INTERFACE I_Singleton

METHOD Message : String
VAR_INPUT
END_VAR
END_METHOD

END_INTERFACE

(* stored: Version 1.1.0.1, ProductVersion 3.1.4024.12
   Itf I_Singleton: Id {a5eba910-5db8-4f2d-a1d3-8e1dad0343dd}
   Method Message: Id {d8f90746-29e8-4fd2-ac8e-814914aeaa76} *)
